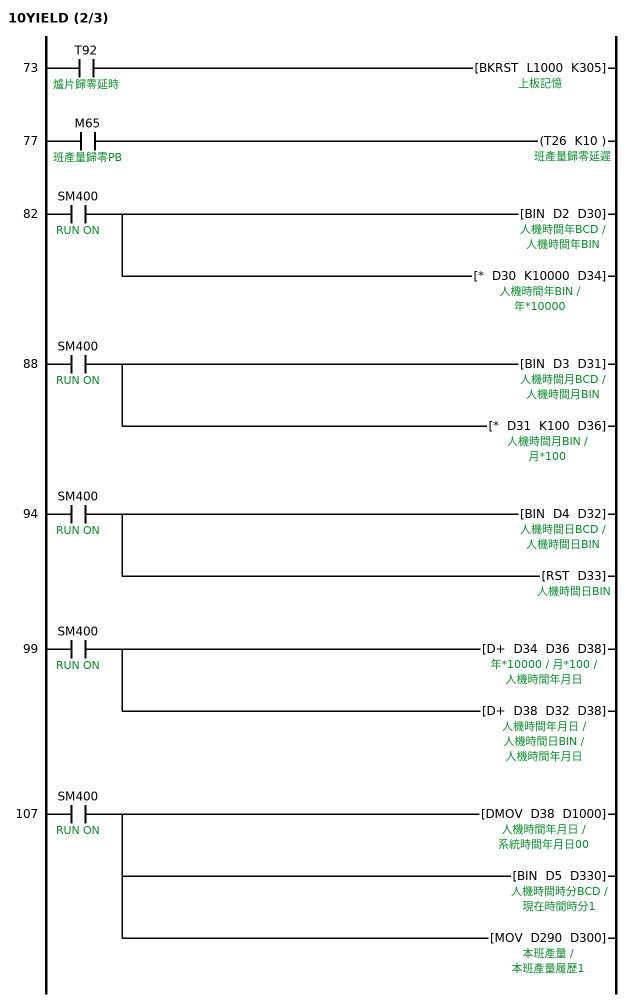
[picture p48: ladder of 10YIELD, rungs at steps 73 to 107]
73    LD      T92  ; 爐片歸零延時
      BKRST   L1000 K305
77    LD      M65  ; 班產量歸零PB
      OUT     T26 K10  ; 班產量歸零延遲
82    LD      SM400  ; RUN ON
      BIN     D2 D30  ; 人機時間年BCD / 人機時間年BIN
      *       D30 K10000 D34  ; 年*10000
88    LD      SM400  ; RUN ON
      BIN     D3 D31  ; 人機時間月BCD / 人機時間月BIN
      *       D31 K100 D36  ; 月*100
94    LD      SM400  ; RUN ON
      BIN     D4 D32  ; 人機時間日BCD / 人機時間日BIN
      RST     D33  ; 人機時間日BIN
99    LD      SM400  ; RUN ON
      D+      D34 D36 D38  ; 人機時間年月日
      D+      D38 D32 D38
107   LD      SM400  ; RUN ON
      DMOV    D38 D1000  ; 系統時間年月日00
      BIN     D5 D330  ; 人機時間時分BCD / 現在時間時分1
      MOV     D290 D300  ; 本班產量履歷1
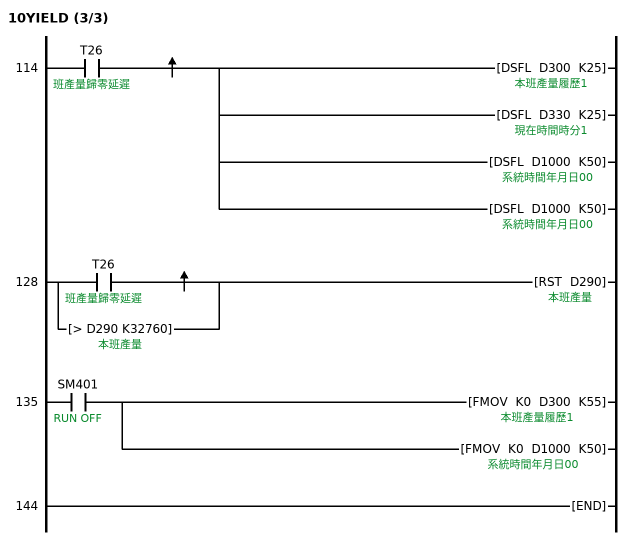
114   LD      T26  ; 班產量歸零延遲
      MEP
      DSFL    D300 K25
      DSFL    D330 K25
      DSFL    D1000 K50
      DSFL    D1000 K50
128   LD      T26  ; 班產量歸零延遲
      MEP
      OR>     D290 K32760  ; 本班產量
      RST     D290  ; 本班產量
135   LD      SM401  ; RUN OFF
      FMOV    K0 D300 K55
      FMOV    K0 D1000 K50
144   END
END_PROGRAM

PROGRAM 11MAINTE
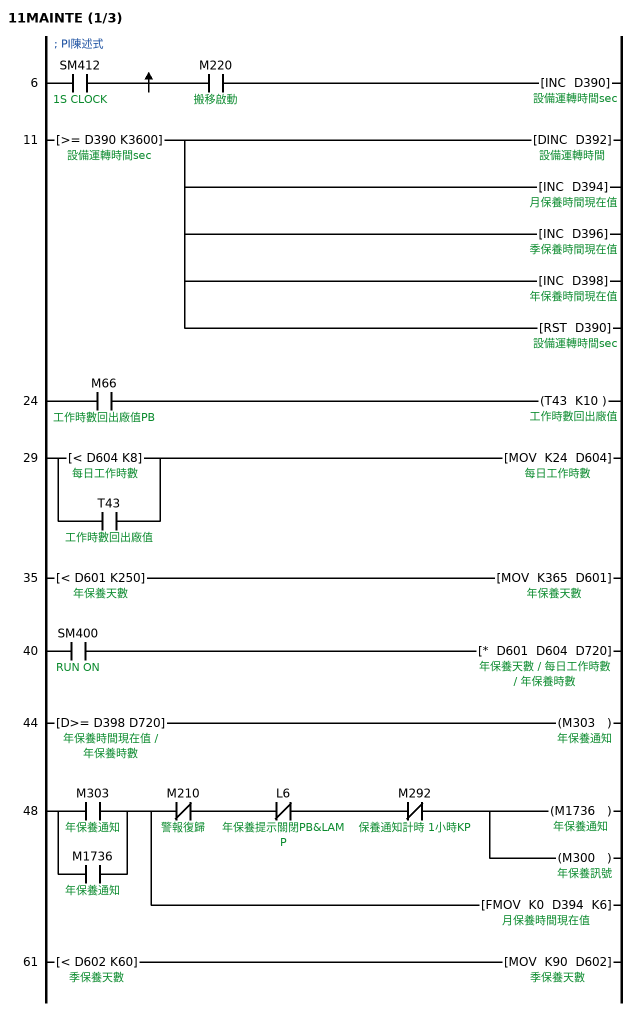
; PI陳述式
6     LD      SM412  ; 1S CLOCK
      MEP
      AND     M220  ; 搬移啟動
      INC     D390  ; 設備運轉時間sec
11    LD>=    D390 K3600  ; 設備運轉時間sec
      DINC    D392  ; 設備運轉時間
      INC     D394  ; 月保養時間現在值
      INC     D396  ; 季保養時間現在值
      INC     D398  ; 年保養時間現在值
      RST     D390  ; 設備運轉時間sec
24    LD      M66  ; 工作時數回出廠值PB
      OUT     T43 K10  ; 工作時數回出廠值
29    LD<     D604 K8  ; 每日工作時數
      OR      T43  ; 工作時數回出廠值
      MOV     K24 D604
35    LD<     D601 K250  ; 年保養天數
      MOV     K365 D601
40    LD      SM400  ; RUN ON
      *       D601 D604 D720  ; 年保養時數
44    LDD>=   D398 D720  ; 年保養時間現在值 / 年保養時數
      OUT     M303  ; 年保養通知
48    LD      M303  ; 年保養通知
      OR      M1736  ; 年保養通知
      MPS
      ANI     M210  ; 警報復歸
      ANI     L6  ; 年保養提示關閉PB&LAMP
      ANI     M292  ; 保養通知計時 1小時KP
      OUT     M1736  ; 年保養通知
      OUT     M300  ; 年保養訊號
      MPP
      FMOV    K0 D394 K6
61    LD<     D602 K60  ; 季保養天數
      MOV     K90 D602
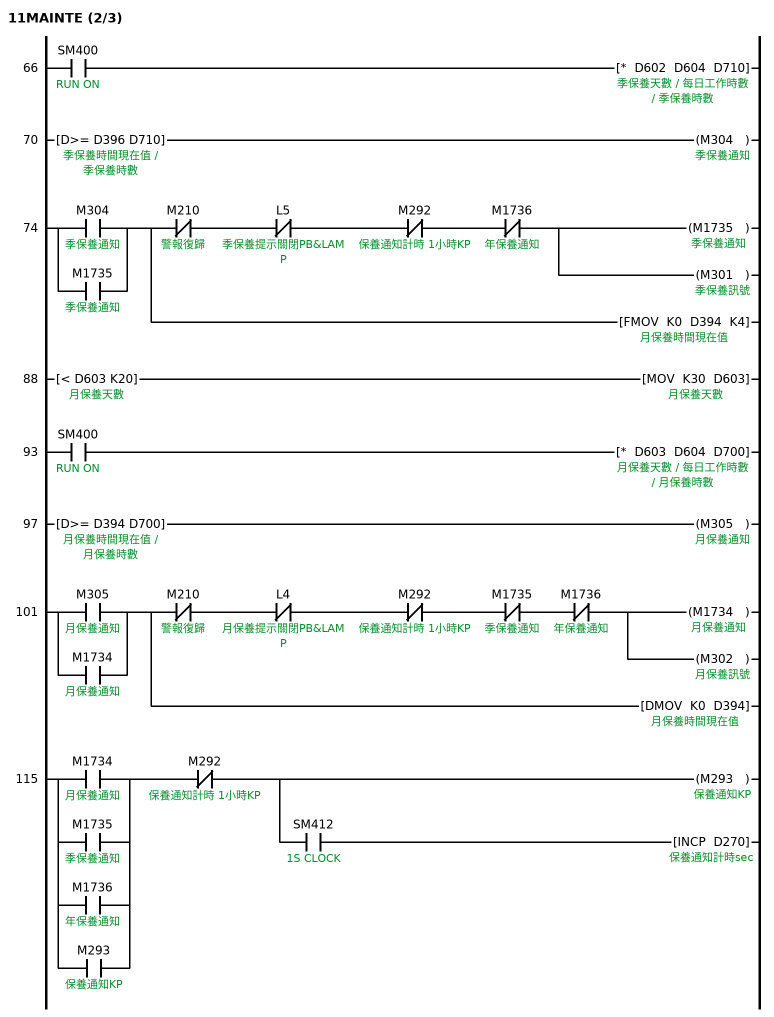
66    LD      SM400  ; RUN ON
      *       D602 D604 D710  ; 季保養時數
70    LDD>=   D396 D710  ; 季保養時間現在值 / 季保養時數
      OUT     M304  ; 季保養通知
74    LD      M304  ; 季保養通知
      OR      M1735  ; 季保養通知
      MPS
      ANI     M210  ; 警報復歸
      ANI     L5  ; 季保養提示關閉PB&LAMP
      ANI     M292  ; 保養通知計時 1小時KP
      ANI     M1736  ; 年保養通知
      OUT     M1735  ; 季保養通知
      OUT     M301  ; 季保養訊號
      MPP
      FMOV    K0 D394 K4
88    LD<     D603 K20  ; 月保養天數
      MOV     K30 D603
93    LD      SM400  ; RUN ON
      *       D603 D604 D700  ; 月保養時數
97    LDD>=   D394 D700  ; 月保養時間現在值 / 月保養時數
      OUT     M305  ; 月保養通知
101   LD      M305  ; 月保養通知
      OR      M1734  ; 月保養通知
      MPS
      ANI     M210  ; 警報復歸
      ANI     L4  ; 月保養提示關閉PB&LAMP
      ANI     M292  ; 保養通知計時 1小時KP
      ANI     M1735  ; 季保養通知
      ANI     M1736  ; 年保養通知
      OUT     M1734  ; 月保養通知
      OUT     M302  ; 月保養訊號
      MPP
      DMOV    K0 D394
115   LD      M1734  ; 月保養通知
      OR      M1735  ; 季保養通知
      OR      M1736  ; 年保養通知
      OR      M293  ; 保養通知KP
      ANI     M292  ; 保養通知計時 1小時KP
      OUT     M293  ; 保養通知KP
      AND     SM412  ; 1S CLOCK
      INCP    D270  ; 保養通知計時sec
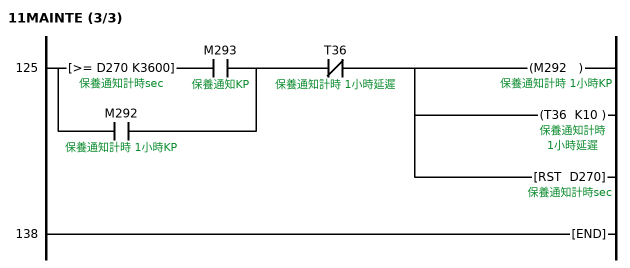
125   LD>=    D270 K3600  ; 保養通知計時sec
      AND     M293  ; 保養通知KP
      OR      M292  ; 保養通知計時 1小時KP
      ANI     T36  ; 保養通知計時 1小時延遲
      OUT     M292  ; 保養通知計時 1小時KP
      OUT     T36 K10  ; 保養通知計時 1小時延遲
      RST     D270  ; 保養通知計時sec
138   END
END_PROGRAM

PROGRAM 12ALARM1
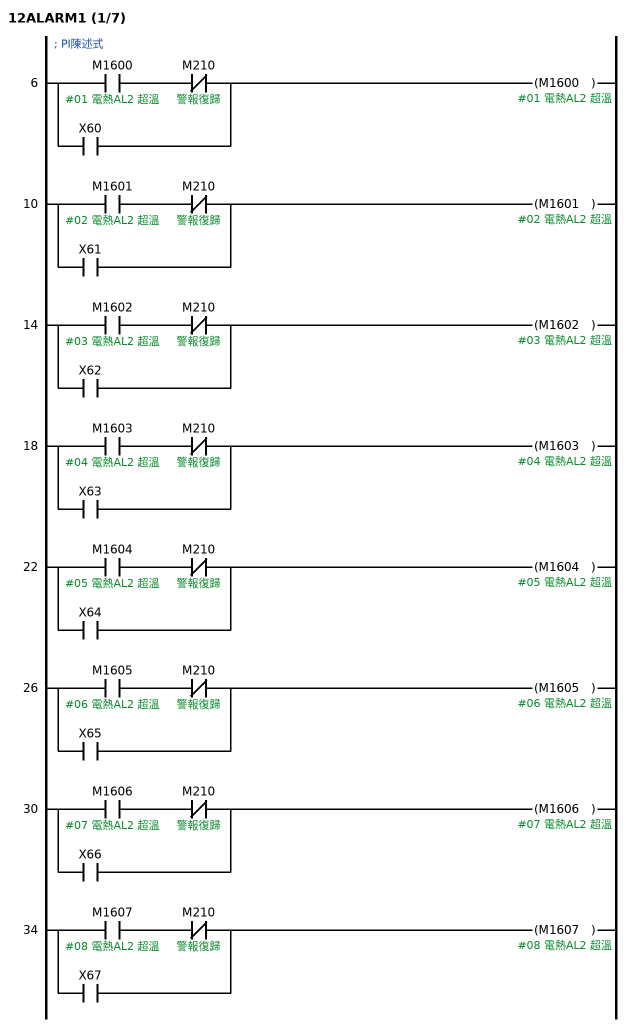
; PI陳述式
6     LD      M1600  ; #01 電熱AL2 超溫
      ANI     M210  ; 警報復歸
      OR      X60
      OUT     M1600  ; #01 電熱AL2 超溫
10    LD      M1601  ; #02 電熱AL2 超溫
      ANI     M210  ; 警報復歸
      OR      X61
      OUT     M1601  ; #02 電熱AL2 超溫
14    LD      M1602  ; #03 電熱AL2 超溫
      ANI     M210  ; 警報復歸
      OR      X62
      OUT     M1602  ; #03 電熱AL2 超溫
18    LD      M1603  ; #04 電熱AL2 超溫
      ANI     M210  ; 警報復歸
      OR      X63
      OUT     M1603  ; #04 電熱AL2 超溫
22    LD      M1604  ; #05 電熱AL2 超溫
      ANI     M210  ; 警報復歸
      OR      X64
      OUT     M1604  ; #05 電熱AL2 超溫
26    LD      M1605  ; #06 電熱AL2 超溫
      ANI     M210  ; 警報復歸
      OR      X65
      OUT     M1605  ; #06 電熱AL2 超溫
30    LD      M1606  ; #07 電熱AL2 超溫
      ANI     M210  ; 警報復歸
      OR      X66
      OUT     M1606  ; #07 電熱AL2 超溫
34    LD      M1607  ; #08 電熱AL2 超溫
      ANI     M210  ; 警報復歸
      OR      X67
      OUT     M1607  ; #08 電熱AL2 超溫
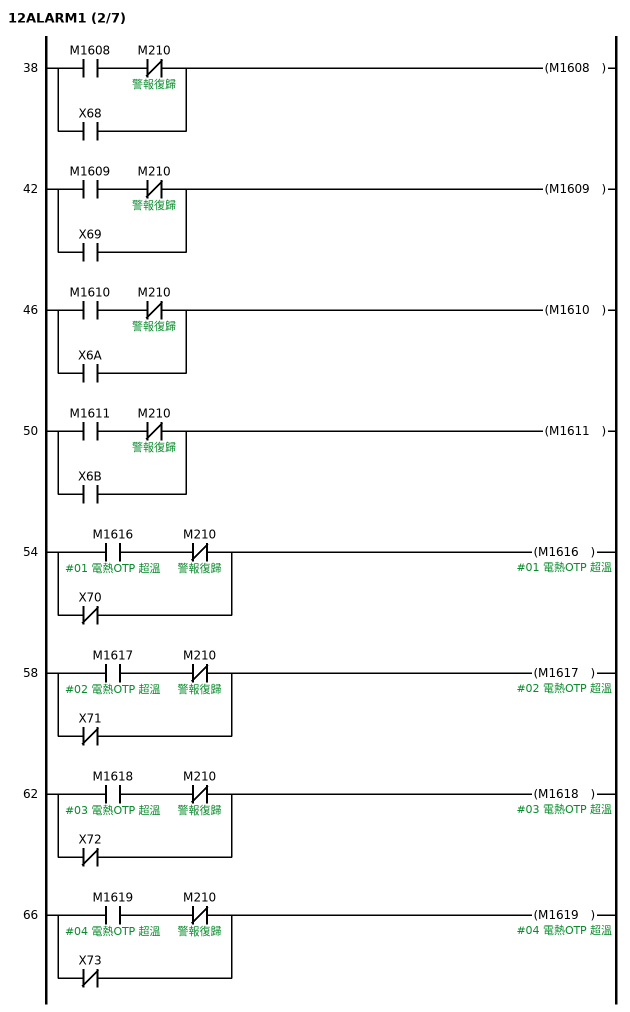
38    LD      M1608
      ANI     M210  ; 警報復歸
      OR      X68
      OUT     M1608
42    LD      M1609
      ANI     M210  ; 警報復歸
      OR      X69
      OUT     M1609
46    LD      M1610
      ANI     M210  ; 警報復歸
      OR      X6A
      OUT     M1610
50    LD      M1611
      ANI     M210  ; 警報復歸
      OR      X6B
      OUT     M1611
54    LD      M1616  ; #01 電熱OTP 超溫
      ANI     M210  ; 警報復歸
      ORI     X70
      OUT     M1616  ; #01 電熱OTP 超溫
58    LD      M1617  ; #02 電熱OTP 超溫
      ANI     M210  ; 警報復歸
      ORI     X71
      OUT     M1617  ; #02 電熱OTP 超溫
62    LD      M1618  ; #03 電熱OTP 超溫
      ANI     M210  ; 警報復歸
      ORI     X72
      OUT     M1618  ; #03 電熱OTP 超溫
66    LD      M1619  ; #04 電熱OTP 超溫
      ANI     M210  ; 警報復歸
      ORI     X73
      OUT     M1619  ; #04 電熱OTP 超溫
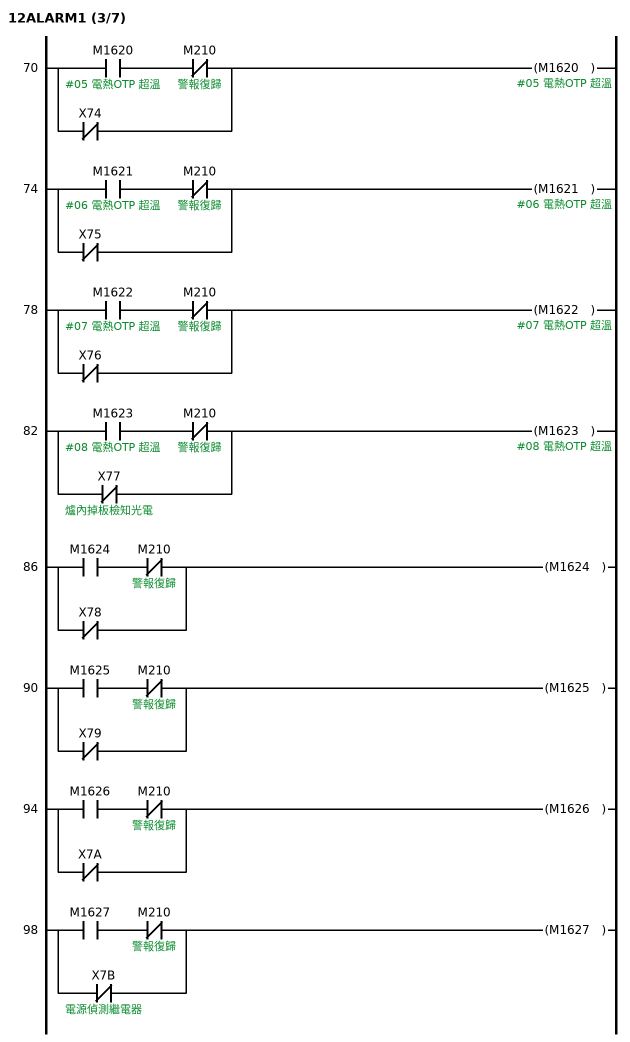
70    LD      M1620  ; #05 電熱OTP 超溫
      ANI     M210  ; 警報復歸
      ORI     X74
      OUT     M1620  ; #05 電熱OTP 超溫
74    LD      M1621  ; #06 電熱OTP 超溫
      ANI     M210  ; 警報復歸
      ORI     X75
      OUT     M1621  ; #06 電熱OTP 超溫
78    LD      M1622  ; #07 電熱OTP 超溫
      ANI     M210  ; 警報復歸
      ORI     X76
      OUT     M1622  ; #07 電熱OTP 超溫
82    LD      M1623  ; #08 電熱OTP 超溫
      ANI     M210  ; 警報復歸
      ORI     X77  ; 爐內掉板檢知光電
      OUT     M1623  ; #08 電熱OTP 超溫
86    LD      M1624
      ANI     M210  ; 警報復歸
      ORI     X78
      OUT     M1624
90    LD      M1625
      ANI     M210  ; 警報復歸
      ORI     X79
      OUT     M1625
94    LD      M1626
      ANI     M210  ; 警報復歸
      ORI     X7A
      OUT     M1626
98    LD      M1627
      ANI     M210  ; 警報復歸
      ORI     X7B  ; 電源偵測繼電器
      OUT     M1627
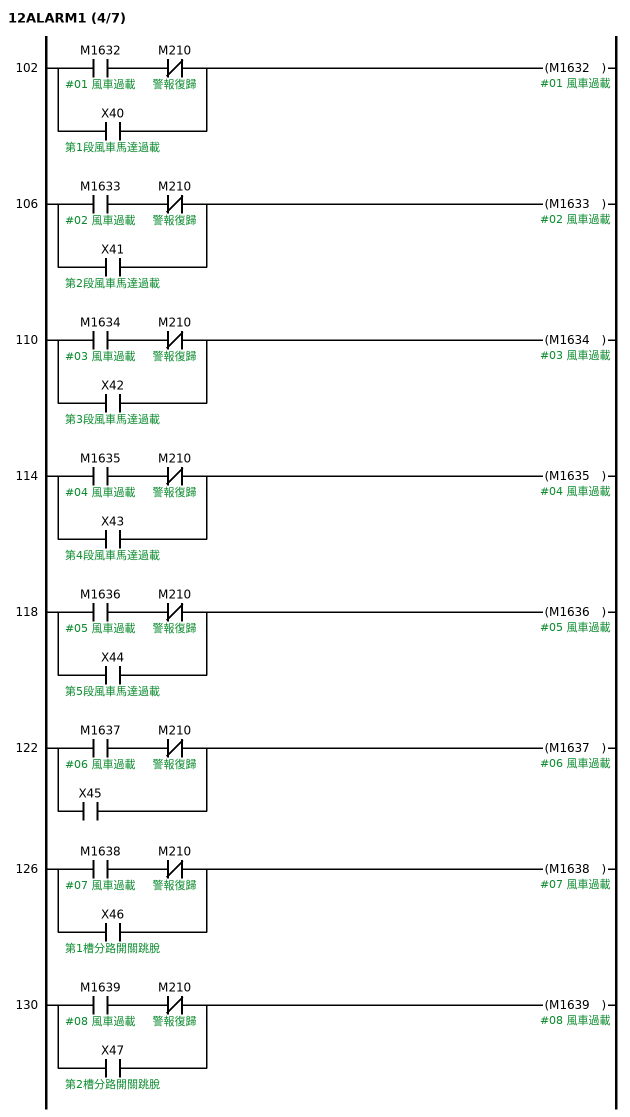
102   LD      M1632  ; #01 風車過載
      ANI     M210  ; 警報復歸
      OR      X40  ; 第1段風車馬達過載
      OUT     M1632  ; #01 風車過載
106   LD      M1633  ; #02 風車過載
      ANI     M210  ; 警報復歸
      OR      X41  ; 第2段風車馬達過載
      OUT     M1633  ; #02 風車過載
110   LD      M1634  ; #03 風車過載
      ANI     M210  ; 警報復歸
      OR      X42  ; 第3段風車馬達過載
      OUT     M1634  ; #03 風車過載
114   LD      M1635  ; #04 風車過載
      ANI     M210  ; 警報復歸
      OR      X43  ; 第4段風車馬達過載
      OUT     M1635  ; #04 風車過載
118   LD      M1636  ; #05 風車過載
      ANI     M210  ; 警報復歸
      OR      X44  ; 第5段風車馬達過載
      OUT     M1636  ; #05 風車過載
122   LD      M1637  ; #06 風車過載
      ANI     M210  ; 警報復歸
      OR      X45
      OUT     M1637  ; #06 風車過載
126   LD      M1638  ; #07 風車過載
      ANI     M210  ; 警報復歸
      OR      X46  ; 第1槽分路開關跳脫
      OUT     M1638  ; #07 風車過載
130   LD      M1639  ; #08 風車過載
      ANI     M210  ; 警報復歸
      OR      X47  ; 第2槽分路開關跳脫
      OUT     M1639  ; #08 風車過載
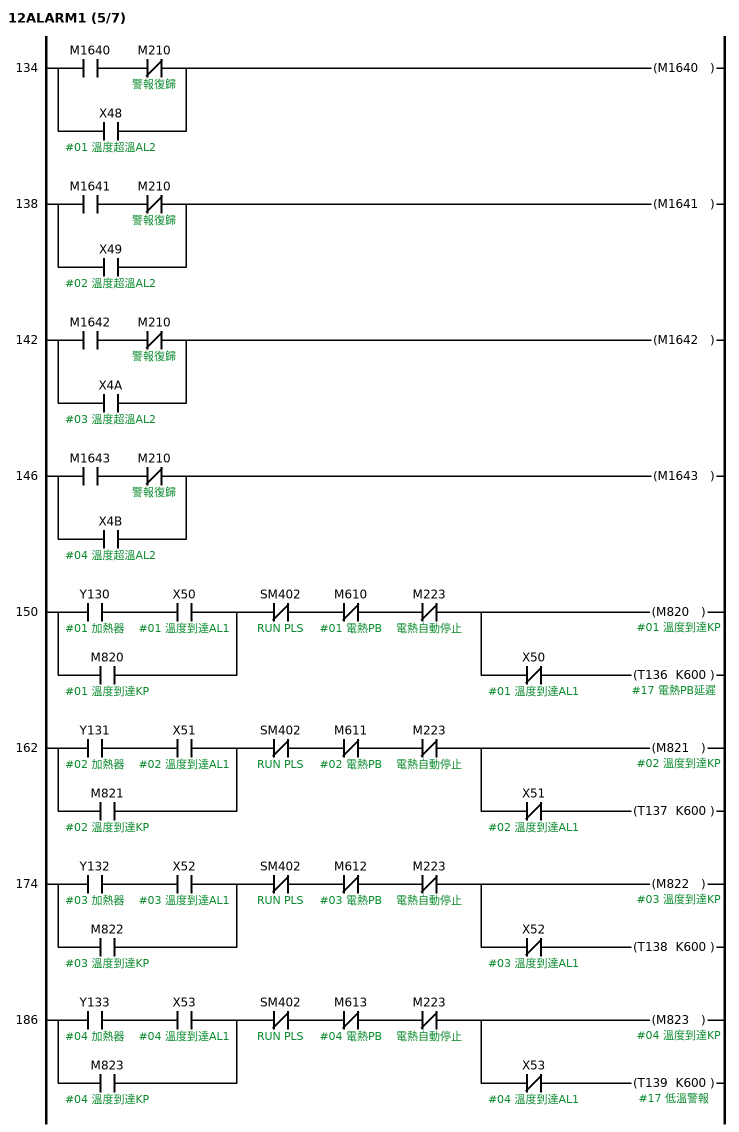
134   LD      M1640
      ANI     M210  ; 警報復歸
      OR      X48  ; #01 溫度超溫AL2
      OUT     M1640
138   LD      M1641
      ANI     M210  ; 警報復歸
      OR      X49  ; #02 溫度超溫AL2
      OUT     M1641
142   LD      M1642
      ANI     M210  ; 警報復歸
      OR      X4A  ; #03 溫度超溫AL2
      OUT     M1642
146   LD      M1643
      ANI     M210  ; 警報復歸
      OR      X4B  ; #04 溫度超溫AL2
      OUT     M1643
150   LD      Y130  ; #01 加熱器
      AND     X50  ; #01 溫度到達AL1
      OR      M820  ; #01 溫度到達KP
      ANI     SM402  ; RUN PLS
      ANI     M610  ; #01 電熱PB
      ANI     M223  ; 電熱自動停止
      OUT     M820  ; #01 溫度到達KP
      ANI     X50  ; #01 溫度到達AL1
      OUT     T136 K600  ; #17 電熱PB延遲
162   LD      Y131  ; #02 加熱器
      AND     X51  ; #02 溫度到達AL1
      OR      M821  ; #02 溫度到達KP
      ANI     SM402  ; RUN PLS
      ANI     M611  ; #02 電熱PB
      ANI     M223  ; 電熱自動停止
      OUT     M821  ; #02 溫度到達KP
      ANI     X51  ; #02 溫度到達AL1
      OUT     T137 K600
174   LD      Y132  ; #03 加熱器
      AND     X52  ; #03 溫度到達AL1
      OR      M822  ; #03 溫度到達KP
      ANI     SM402  ; RUN PLS
      ANI     M612  ; #03 電熱PB
      ANI     M223  ; 電熱自動停止
      OUT     M822  ; #03 溫度到達KP
      ANI     X52  ; #03 溫度到達AL1
      OUT     T138 K600
186   LD      Y133  ; #04 加熱器
      AND     X53  ; #04 溫度到達AL1
      OR      M823  ; #04 溫度到達KP
      ANI     SM402  ; RUN PLS
      ANI     M613  ; #04 電熱PB
      ANI     M223  ; 電熱自動停止
      OUT     M823  ; #04 溫度到達KP
      ANI     X53  ; #04 溫度到達AL1
      OUT     T139 K600  ; #17 低溫警報
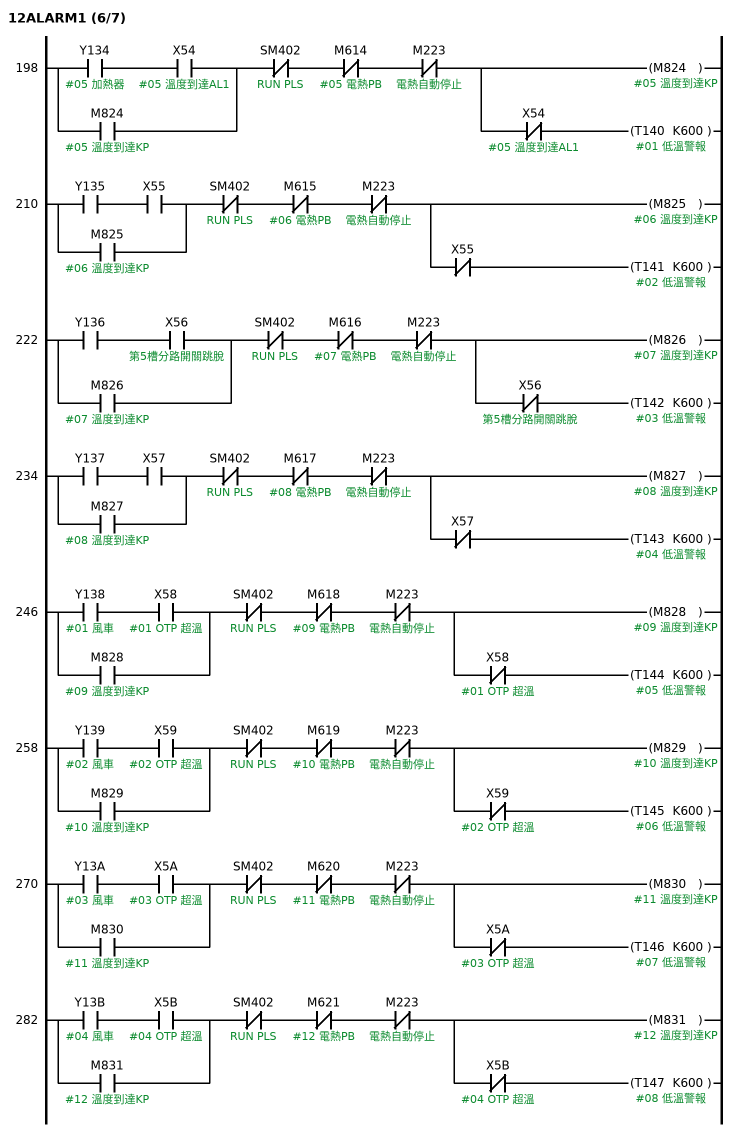
198   LD      Y134  ; #05 加熱器
      AND     X54  ; #05 溫度到達AL1
      OR      M824  ; #05 溫度到達KP
      ANI     SM402  ; RUN PLS
      ANI     M614  ; #05 電熱PB
      ANI     M223  ; 電熱自動停止
      OUT     M824  ; #05 溫度到達KP
      ANI     X54  ; #05 溫度到達AL1
      OUT     T140 K600  ; #01 低溫警報
210   LD      Y135
      AND     X55
      OR      M825  ; #06 溫度到達KP
      ANI     SM402  ; RUN PLS
      ANI     M615  ; #06 電熱PB
      ANI     M223  ; 電熱自動停止
      OUT     M825  ; #06 溫度到達KP
      ANI     X55
      OUT     T141 K600  ; #02 低溫警報
222   LD      Y136
      AND     X56  ; 第5槽分路開關跳脫
      OR      M826  ; #07 溫度到達KP
      ANI     SM402  ; RUN PLS
      ANI     M616  ; #07 電熱PB
      ANI     M223  ; 電熱自動停止
      OUT     M826  ; #07 溫度到達KP
      ANI     X56  ; 第5槽分路開關跳脫
      OUT     T142 K600  ; #03 低溫警報
234   LD      Y137
      AND     X57
      OR      M827  ; #08 溫度到達KP
      ANI     SM402  ; RUN PLS
      ANI     M617  ; #08 電熱PB
      ANI     M223  ; 電熱自動停止
      OUT     M827  ; #08 溫度到達KP
      ANI     X57
      OUT     T143 K600  ; #04 低溫警報
246   LD      Y138  ; #01 風車
      AND     X58  ; #01 OTP 超溫
      OR      M828  ; #09 溫度到達KP
      ANI     SM402  ; RUN PLS
      ANI     M618  ; #09 電熱PB
      ANI     M223  ; 電熱自動停止
      OUT     M828  ; #09 溫度到達KP
      ANI     X58  ; #01 OTP 超溫
      OUT     T144 K600  ; #05 低溫警報
258   LD      Y139  ; #02 風車
      AND     X59  ; #02 OTP 超溫
      OR      M829  ; #10 溫度到達KP
      ANI     SM402  ; RUN PLS
      ANI     M619  ; #10 電熱PB
      ANI     M223  ; 電熱自動停止
      OUT     M829  ; #10 溫度到達KP
      ANI     X59  ; #02 OTP 超溫
      OUT     T145 K600  ; #06 低溫警報
270   LD      Y13A  ; #03 風車
      AND     X5A  ; #03 OTP 超溫
      OR      M830  ; #11 溫度到達KP
      ANI     SM402  ; RUN PLS
      ANI     M620  ; #11 電熱PB
      ANI     M223  ; 電熱自動停止
      OUT     M830  ; #11 溫度到達KP
      ANI     X5A  ; #03 OTP 超溫
      OUT     T146 K600  ; #07 低溫警報
282   LD      Y13B  ; #04 風車
      AND     X5B  ; #04 OTP 超溫
      OR      M831  ; #12 溫度到達KP
      ANI     SM402  ; RUN PLS
      ANI     M621  ; #12 電熱PB
      ANI     M223  ; 電熱自動停止
      OUT     M831  ; #12 溫度到達KP
      ANI     X5B  ; #04 OTP 超溫
      OUT     T147 K600  ; #08 低溫警報
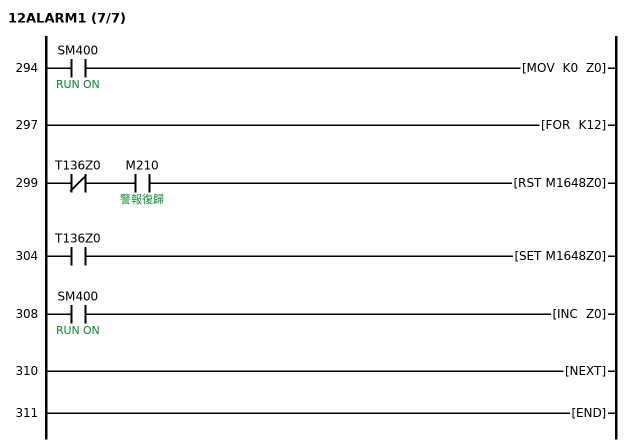
294   LD      SM400  ; RUN ON
      MOV     K0 Z0
297   FOR     K12
299   LDI     T136Z0
      AND     M210  ; 警報復歸
      RST     M1648Z0
304   LD      T136Z0
      SET     M1648Z0
308   LD      SM400  ; RUN ON
      INC     Z0
310   NEXT
311   END
END_PROGRAM

PROGRAM 13ALARM2
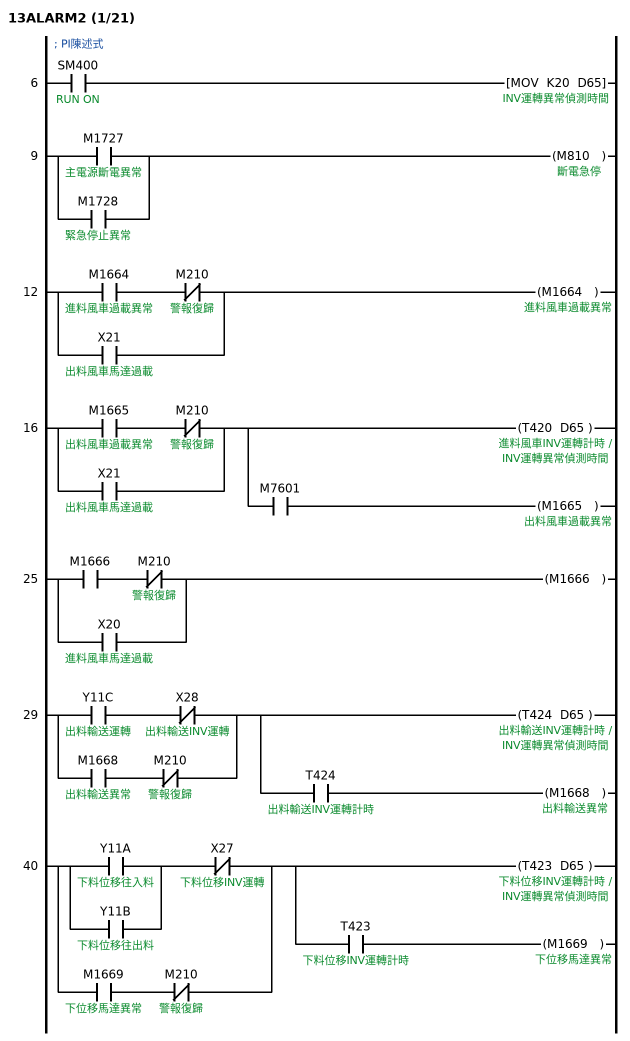
; PI陳述式
6     LD      SM400  ; RUN ON
      MOV     K20 D65  ; INV運轉異常偵測時間
9     LD      M1727  ; 主電源斷電異常
      OR      M1728  ; 緊急停止異常
      OUT     M810  ; 斷電急停
12    LD      M1664  ; 進料風車過載異常
      ANI     M210  ; 警報復歸
      OR      X21  ; 出料風車馬達過載
      OUT     M1664  ; 進料風車過載異常
16    LD      M1665  ; 出料風車過載異常
      ANI     M210  ; 警報復歸
      OR      X21  ; 出料風車馬達過載
      OUT     T420 D65  ; 進料風車INV運轉計時 / INV運轉異常偵測時間
      AND     M7601
      OUT     M1665  ; 出料風車過載異常
25    LD      M1666
      ANI     M210  ; 警報復歸
      OR      X20  ; 進料風車馬達過載
      OUT     M1666
29    LD      Y11C  ; 出料輸送運轉
      ANI     X28  ; 出料輸送INV運轉
      LD      M1668  ; 出料輸送異常
      ANI     M210  ; 警報復歸
      ORB
      OUT     T424 D65  ; 出料輸送INV運轉計時 / INV運轉異常偵測時間
      AND     T424  ; 出料輸送INV運轉計時
      OUT     M1668  ; 出料輸送異常
40    LD      Y11A  ; 下料位移往入料
      OR      Y11B  ; 下料位移往出料
      ANI     X27  ; 下料位移INV運轉
      LD      M1669  ; 下位移馬達異常
      ANI     M210  ; 警報復歸
      ORB
      OUT     T423 D65  ; 下料位移INV運轉計時 / INV運轉異常偵測時間
      AND     T423  ; 下料位移INV運轉計時
      OUT     M1669  ; 下位移馬達異常
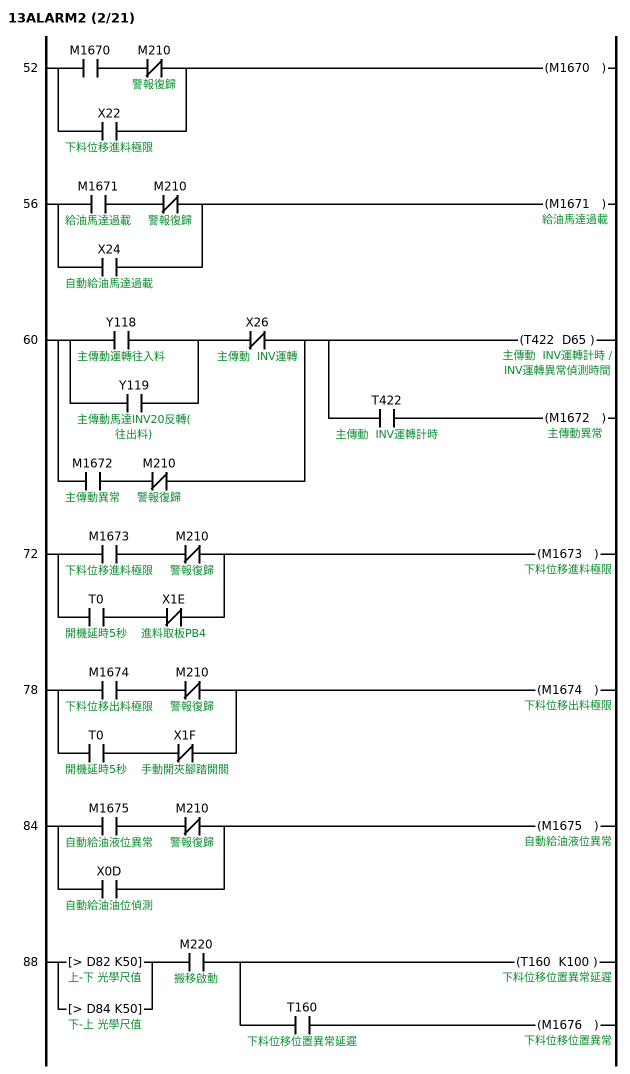
52    LD      M1670
      ANI     M210  ; 警報復歸
      OR      X22  ; 下料位移進料極限
      OUT     M1670
56    LD      M1671  ; 給油馬達過載
      ANI     M210  ; 警報復歸
      OR      X24  ; 自動給油馬達過載
      OUT     M1671  ; 給油馬達過載
60    LD      Y118  ; 主傳動運轉往入料
      OR      Y119  ; 主傳動馬達INV20反轉(往出料)
      ANI     X26  ; 主傳動  INV運轉
      LD      M1672  ; 主傳動異常
      ANI     M210  ; 警報復歸
      ORB
      OUT     T422 D65  ; 主傳動  INV運轉計時 / INV運轉異常偵測時間
      AND     T422  ; 主傳動  INV運轉計時
      OUT     M1672  ; 主傳動異常
72    LD      M1673  ; 下料位移進料極限
      ANI     M210  ; 警報復歸
      LD      T0  ; 開機延時5秒
      ANI     X1E  ; 進料取板PB4
      ORB
      OUT     M1673  ; 下料位移進料極限
78    LD      M1674  ; 下料位移出料極限
      ANI     M210  ; 警報復歸
      LD      T0  ; 開機延時5秒
      ANI     X1F  ; 手動開夾腳踏開關
      ORB
      OUT     M1674  ; 下料位移出料極限
84    LD      M1675  ; 自動給油液位異常
      ANI     M210  ; 警報復歸
      OR      X0D  ; 自動給油油位偵測
      OUT     M1675  ; 自動給油液位異常
88    LD>     D82 K50  ; 上-下 光學尺值
      OR>     D84 K50  ; 下-上 光學尺值
      AND     M220  ; 搬移啟動
      OUT     T160 K100  ; 下料位移位置異常延遲
      AND     T160  ; 下料位移位置異常延遲
      OUT     M1676  ; 下料位移位置異常
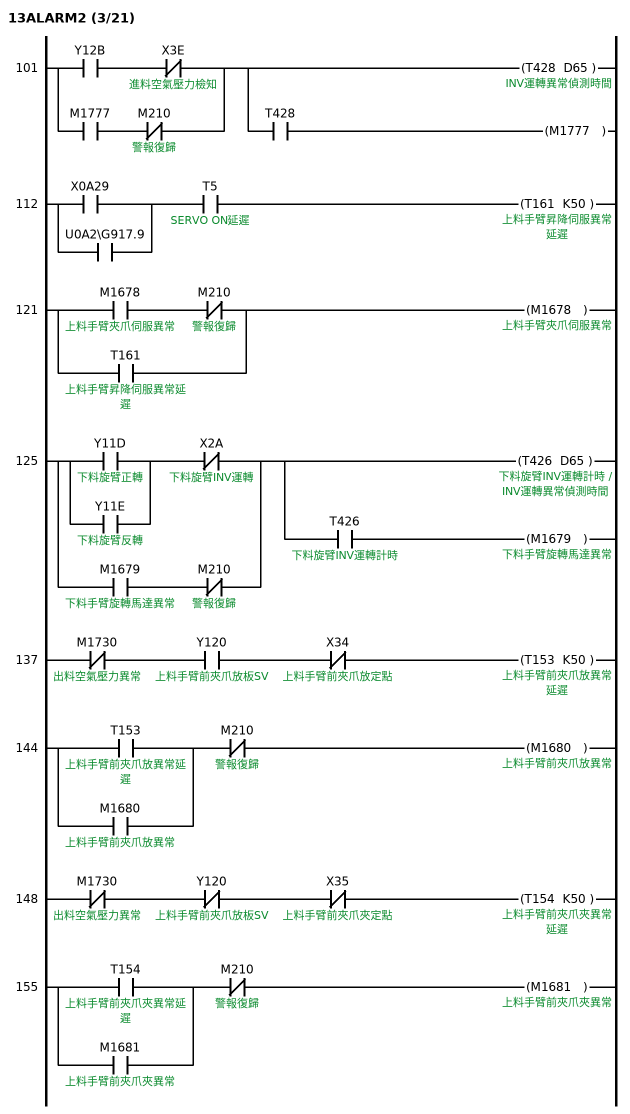
101   LD      Y12B
      ANI     X3E  ; 進料空氣壓力檢知
      LD      M1777
      ANI     M210  ; 警報復歸
      ORB
      OUT     T428 D65  ; INV運轉異常偵測時間
      AND     T428
      OUT     M1777
112   LD      X0A29
      OR      U0A2\G917.9
      AND     T5  ; SERVO ON延遲
      OUT     T161 K50  ; 上料手臂昇降伺服異常延遲
121   LD      M1678  ; 上料手臂夾爪伺服異常
      ANI     M210  ; 警報復歸
      OR      T161  ; 上料手臂昇降伺服異常延遲
      OUT     M1678  ; 上料手臂夾爪伺服異常
125   LD      Y11D  ; 下料旋臂正轉
      OR      Y11E  ; 下料旋臂反轉
      ANI     X2A  ; 下料旋臂INV運轉
      LD      M1679  ; 下料手臂旋轉馬達異常
      ANI     M210  ; 警報復歸
      ORB
      OUT     T426 D65  ; 下料旋臂INV運轉計時 / INV運轉異常偵測時間
      AND     T426  ; 下料旋臂INV運轉計時
      OUT     M1679  ; 下料手臂旋轉馬達異常
137   LDI     M1730  ; 出料空氣壓力異常
      AND     Y120  ; 上料手臂前夾爪放板SV
      ANI     X34  ; 上料手臂前夾爪放定點
      OUT     T153 K50  ; 上料手臂前夾爪放異常延遲
144   LD      T153  ; 上料手臂前夾爪放異常延遲
      OR      M1680  ; 上料手臂前夾爪放異常
      ANI     M210  ; 警報復歸
      OUT     M1680  ; 上料手臂前夾爪放異常
148   LDI     M1730  ; 出料空氣壓力異常
      ANI     Y120  ; 上料手臂前夾爪放板SV
      ANI     X35  ; 上料手臂前夾爪夾定點
      OUT     T154 K50  ; 上料手臂前夾爪夾異常延遲
155   LD      T154  ; 上料手臂前夾爪夾異常延遲
      OR      M1681  ; 上料手臂前夾爪夾異常
      ANI     M210  ; 警報復歸
      OUT     M1681  ; 上料手臂前夾爪夾異常
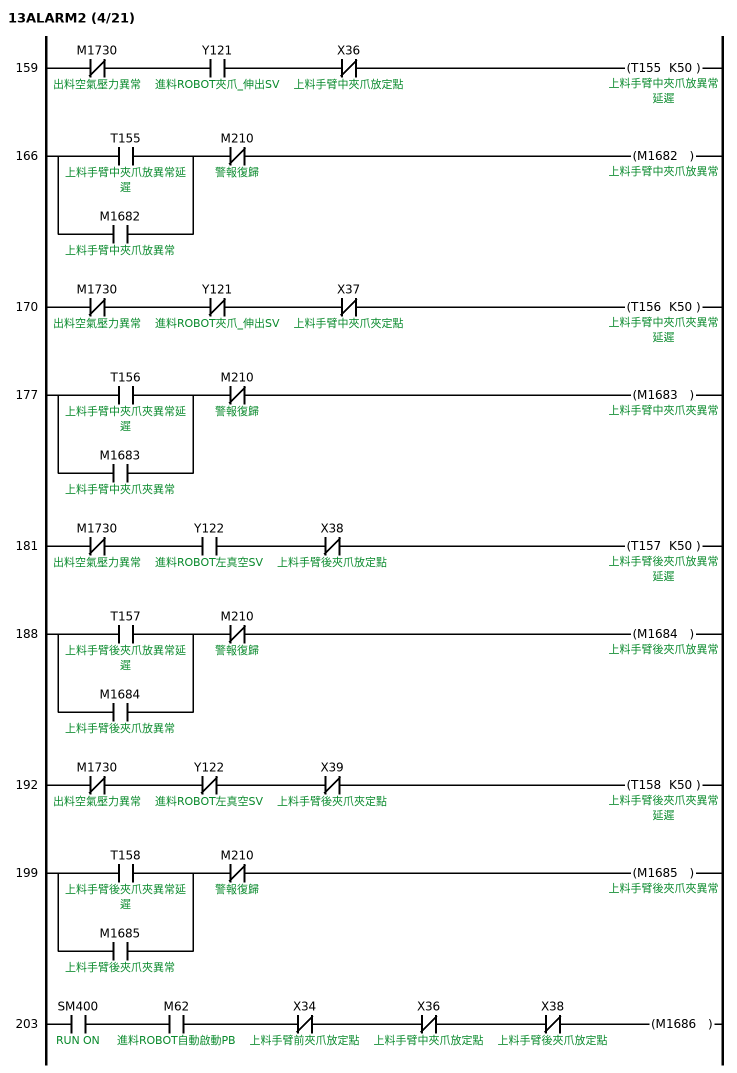
159   LDI     M1730  ; 出料空氣壓力異常
      AND     Y121  ; 進料ROBOT夾爪_伸出SV
      ANI     X36  ; 上料手臂中夾爪放定點
      OUT     T155 K50  ; 上料手臂中夾爪放異常延遲
166   LD      T155  ; 上料手臂中夾爪放異常延遲
      OR      M1682  ; 上料手臂中夾爪放異常
      ANI     M210  ; 警報復歸
      OUT     M1682  ; 上料手臂中夾爪放異常
170   LDI     M1730  ; 出料空氣壓力異常
      ANI     Y121  ; 進料ROBOT夾爪_伸出SV
      ANI     X37  ; 上料手臂中夾爪夾定點
      OUT     T156 K50  ; 上料手臂中夾爪夾異常延遲
177   LD      T156  ; 上料手臂中夾爪夾異常延遲
      OR      M1683  ; 上料手臂中夾爪夾異常
      ANI     M210  ; 警報復歸
      OUT     M1683  ; 上料手臂中夾爪夾異常
181   LDI     M1730  ; 出料空氣壓力異常
      AND     Y122  ; 進料ROBOT左真空SV
      ANI     X38  ; 上料手臂後夾爪放定點
      OUT     T157 K50  ; 上料手臂後夾爪放異常延遲
188   LD      T157  ; 上料手臂後夾爪放異常延遲
      OR      M1684  ; 上料手臂後夾爪放異常
      ANI     M210  ; 警報復歸
      OUT     M1684  ; 上料手臂後夾爪放異常
192   LDI     M1730  ; 出料空氣壓力異常
      ANI     Y122  ; 進料ROBOT左真空SV
      ANI     X39  ; 上料手臂後夾爪夾定點
      OUT     T158 K50  ; 上料手臂後夾爪夾異常延遲
199   LD      T158  ; 上料手臂後夾爪夾異常延遲
      OR      M1685  ; 上料手臂後夾爪夾異常
      ANI     M210  ; 警報復歸
      OUT     M1685  ; 上料手臂後夾爪夾異常
203   LD      SM400  ; RUN ON
      AND     M62  ; 進料ROBOT自動啟動PB
      ANI     X34  ; 上料手臂前夾爪放定點
      ANI     X36  ; 上料手臂中夾爪放定點
      ANI     X38  ; 上料手臂後夾爪放定點
      OUT     M1686
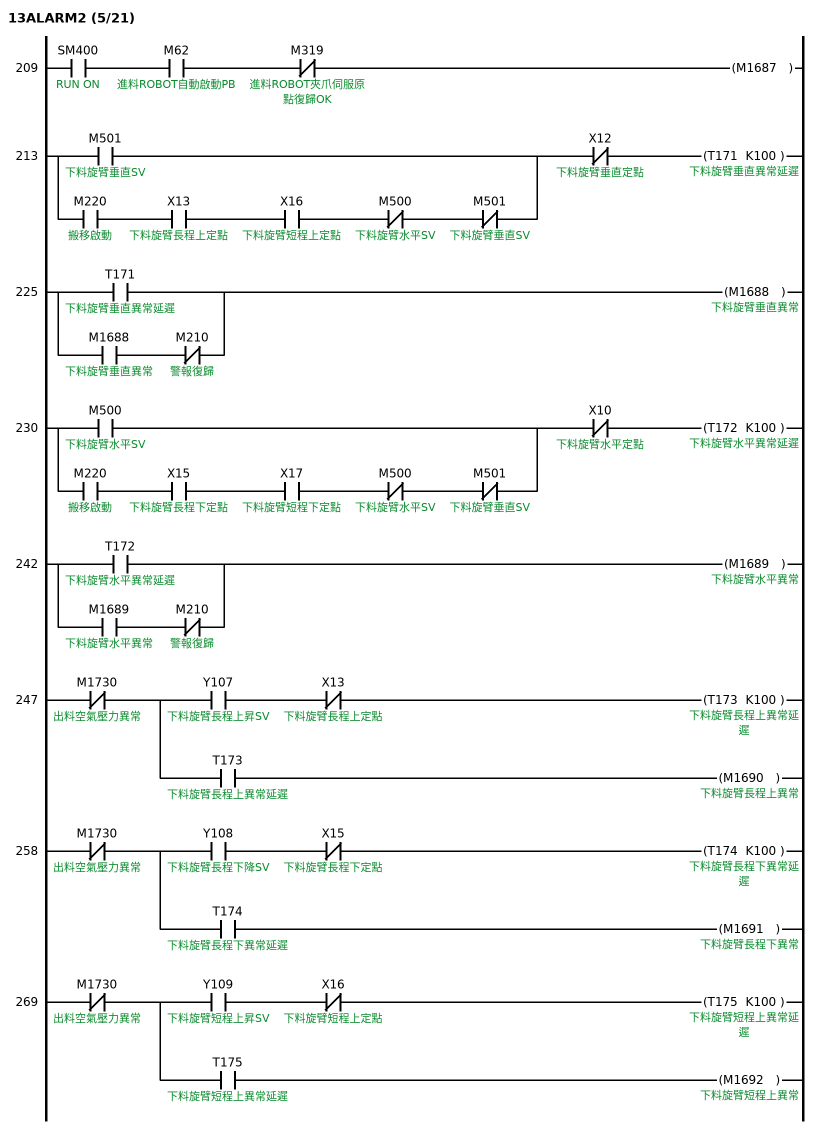
209   LD      SM400  ; RUN ON
      AND     M62  ; 進料ROBOT自動啟動PB
      ANI     M319  ; 進料ROBOT夾爪伺服原點復歸OK
      OUT     M1687
213   LD      M501  ; 下料旋臂垂直SV
      LD      M220  ; 搬移啟動
      AND     X13  ; 下料旋臂長程上定點
      AND     X16  ; 下料旋臂短程上定點
      ANI     M500  ; 下料旋臂水平SV
      ANI     M501  ; 下料旋臂垂直SV
      ORB
      ANI     X12  ; 下料旋臂垂直定點
      OUT     T171 K100  ; 下料旋臂垂直異常延遲
225   LD      T171  ; 下料旋臂垂直異常延遲
      LD      M1688  ; 下料旋臂垂直異常
      ANI     M210  ; 警報復歸
      ORB
      OUT     M1688  ; 下料旋臂垂直異常
230   LD      M500  ; 下料旋臂水平SV
      LD      M220  ; 搬移啟動
      AND     X15  ; 下料旋臂長程下定點
      AND     X17  ; 下料旋臂短程下定點
      ANI     M500  ; 下料旋臂水平SV
      ANI     M501  ; 下料旋臂垂直SV
      ORB
      ANI     X10  ; 下料旋臂水平定點
      OUT     T172 K100  ; 下料旋臂水平異常延遲
242   LD      T172  ; 下料旋臂水平異常延遲
      LD      M1689  ; 下料旋臂水平異常
      ANI     M210  ; 警報復歸
      ORB
      OUT     M1689  ; 下料旋臂水平異常
247   LDI     M1730  ; 出料空氣壓力異常
      MPS
      AND     Y107  ; 下料旋臂長程上昇SV
      ANI     X13  ; 下料旋臂長程上定點
      OUT     T173 K100  ; 下料旋臂長程上異常延遲
      MPP
      AND     T173  ; 下料旋臂長程上異常延遲
      OUT     M1690  ; 下料旋臂長程上異常
258   LDI     M1730  ; 出料空氣壓力異常
      MPS
      AND     Y108  ; 下料旋臂長程下降SV
      ANI     X15  ; 下料旋臂長程下定點
      OUT     T174 K100  ; 下料旋臂長程下異常延遲
      MPP
      AND     T174  ; 下料旋臂長程下異常延遲
      OUT     M1691  ; 下料旋臂長程下異常
269   LDI     M1730  ; 出料空氣壓力異常
      MPS
      AND     Y109  ; 下料旋臂短程上昇SV
      ANI     X16  ; 下料旋臂短程上定點
      OUT     T175 K100  ; 下料旋臂短程上異常延遲
      MPP
      AND     T175  ; 下料旋臂短程上異常延遲
      OUT     M1692  ; 下料旋臂短程上異常
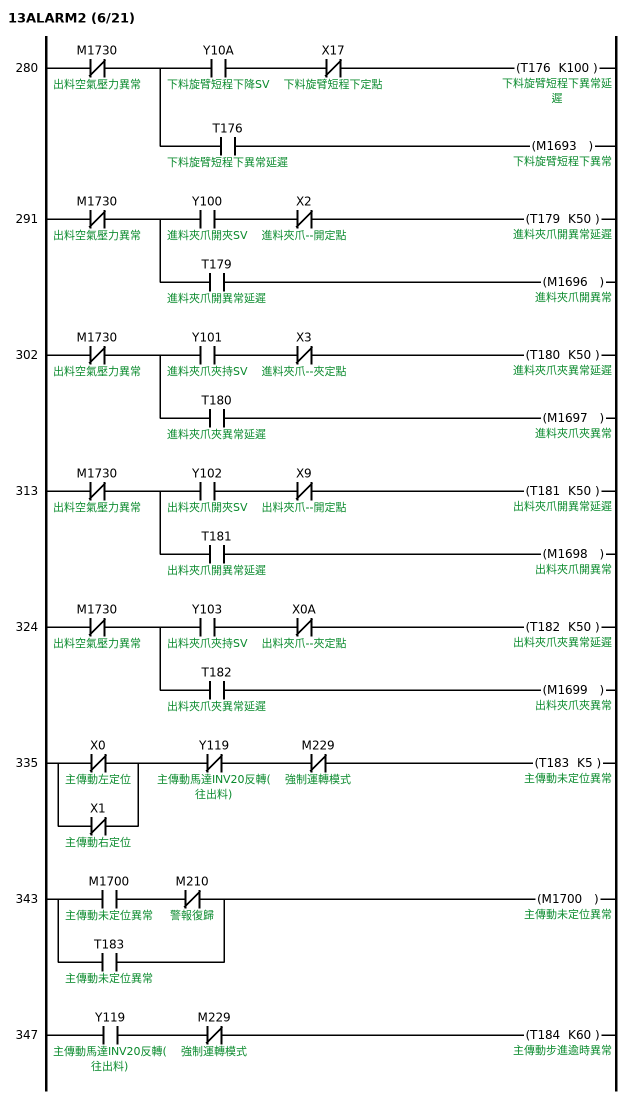
280   LDI     M1730  ; 出料空氣壓力異常
      MPS
      AND     Y10A  ; 下料旋臂短程下降SV
      ANI     X17  ; 下料旋臂短程下定點
      OUT     T176 K100  ; 下料旋臂短程下異常延遲
      MPP
      AND     T176  ; 下料旋臂短程下異常延遲
      OUT     M1693  ; 下料旋臂短程下異常
291   LDI     M1730  ; 出料空氣壓力異常
      MPS
      AND     Y100  ; 進料夾爪開夾SV
      ANI     X2  ; 進料夾爪--開定點
      OUT     T179 K50  ; 進料夾爪開異常延遲
      MPP
      AND     T179  ; 進料夾爪開異常延遲
      OUT     M1696  ; 進料夾爪開異常
302   LDI     M1730  ; 出料空氣壓力異常
      MPS
      AND     Y101  ; 進料夾爪夾持SV
      ANI     X3  ; 進料夾爪--夾定點
      OUT     T180 K50  ; 進料夾爪夾異常延遲
      MPP
      AND     T180  ; 進料夾爪夾異常延遲
      OUT     M1697  ; 進料夾爪夾異常
313   LDI     M1730  ; 出料空氣壓力異常
      MPS
      AND     Y102  ; 出料夾爪開夾SV
      ANI     X9  ; 出料夾爪--開定點
      OUT     T181 K50  ; 出料夾爪開異常延遲
      MPP
      AND     T181  ; 出料夾爪開異常延遲
      OUT     M1698  ; 出料夾爪開異常
324   LDI     M1730  ; 出料空氣壓力異常
      MPS
      AND     Y103  ; 出料夾爪夾持SV
      ANI     X0A  ; 出料夾爪--夾定點
      OUT     T182 K50  ; 出料夾爪夾異常延遲
      MPP
      AND     T182  ; 出料夾爪夾異常延遲
      OUT     M1699  ; 出料夾爪夾異常
335   LDI     X0  ; 主傳動左定位
      ORI     X1  ; 主傳動右定位
      ANI     Y119  ; 主傳動馬達INV20反轉(往出料)
      ANI     M229  ; 強制運轉模式
      OUT     T183 K5  ; 主傳動未定位異常
343   LD      M1700  ; 主傳動未定位異常
      ANI     M210  ; 警報復歸
      OR      T183  ; 主傳動未定位異常
      OUT     M1700  ; 主傳動未定位異常
347   LD      Y119  ; 主傳動馬達INV20反轉(往出料)
      ANI     M229  ; 強制運轉模式
      OUT     T184 K60  ; 主傳動步進逾時異常
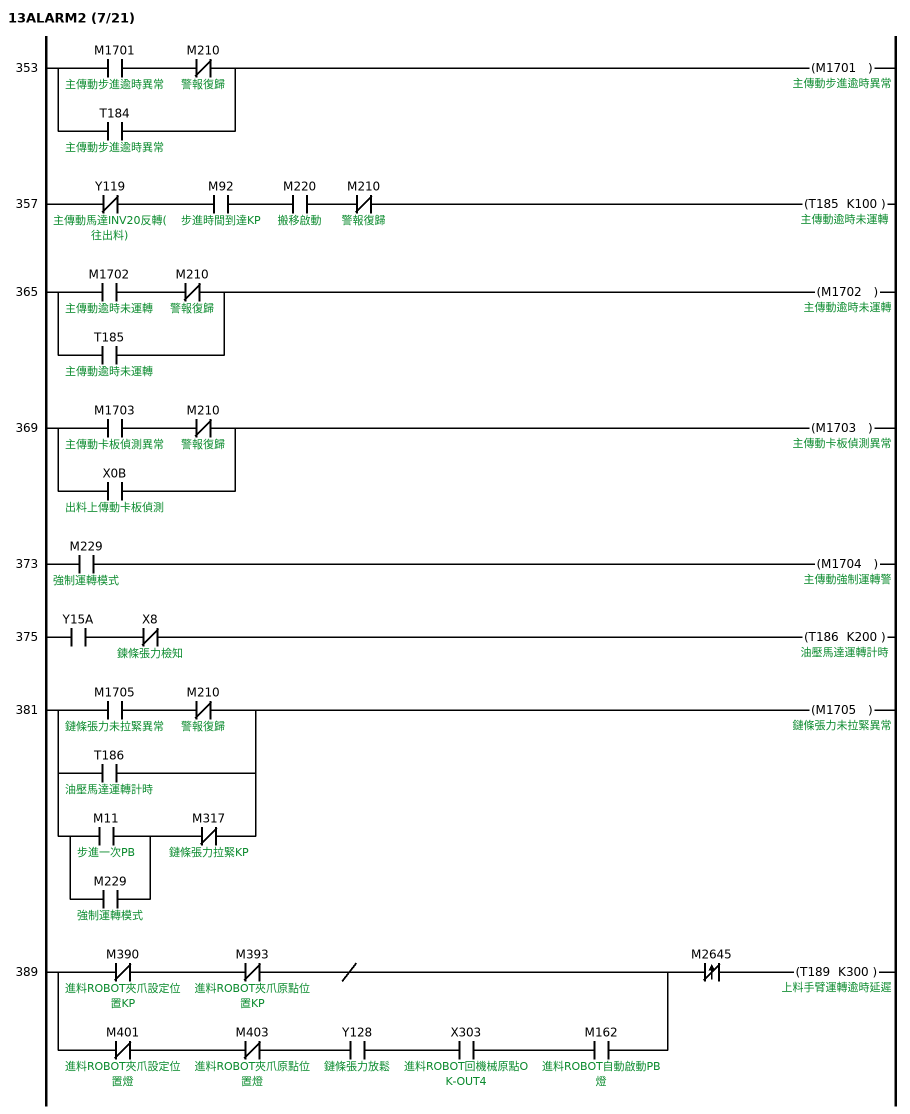
353   LD      M1701  ; 主傳動步進逾時異常
      ANI     M210  ; 警報復歸
      OR      T184  ; 主傳動步進逾時異常
      OUT     M1701  ; 主傳動步進逾時異常
357   LDI     Y119  ; 主傳動馬達INV20反轉(往出料)
      AND     M92  ; 步進時間到達KP
      AND     M220  ; 搬移啟動
      ANI     M210  ; 警報復歸
      OUT     T185 K100  ; 主傳動逾時未運轉
365   LD      M1702  ; 主傳動逾時未運轉
      ANI     M210  ; 警報復歸
      OR      T185  ; 主傳動逾時未運轉
      OUT     M1702  ; 主傳動逾時未運轉
369   LD      M1703  ; 主傳動卡板偵測異常
      ANI     M210  ; 警報復歸
      OR      X0B  ; 出料上傳動卡板偵測
      OUT     M1703  ; 主傳動卡板偵測異常
373   LD      M229  ; 強制運轉模式
      OUT     M1704  ; 主傳動強制運轉警
375   LD      Y15A
      ANI     X8  ; 鍊條張力檢知
      OUT     T186 K200  ; 油壓馬達運轉計時
381   LD      M1705  ; 鏈條張力未拉緊異常
      ANI     M210  ; 警報復歸
      OR      T186  ; 油壓馬達運轉計時
      LD      M11  ; 步進一次PB
      OR      M229  ; 強制運轉模式
      ANI     M317  ; 鏈條張力拉緊KP
      ORB
      OUT     M1705  ; 鏈條張力未拉緊異常
389   LDI     M390  ; 進料ROBOT夾爪設定位置KP
      ANI     M393  ; 進料ROBOT夾爪原點位置KP
      INV
      LDI     M401  ; 進料ROBOT夾爪設定位置燈
      ANI     M403  ; 進料ROBOT夾爪原點位置燈
      AND     Y128  ; 鏈條張力放鬆
      AND     X303  ; 進料ROBOT回機械原點OK-OUT4
      AND     M162  ; 進料ROBOT自動啟動PB燈
      ORB
      ANDPI   M2645
      OUT     T189 K300  ; 上料手臂運轉逾時延遲
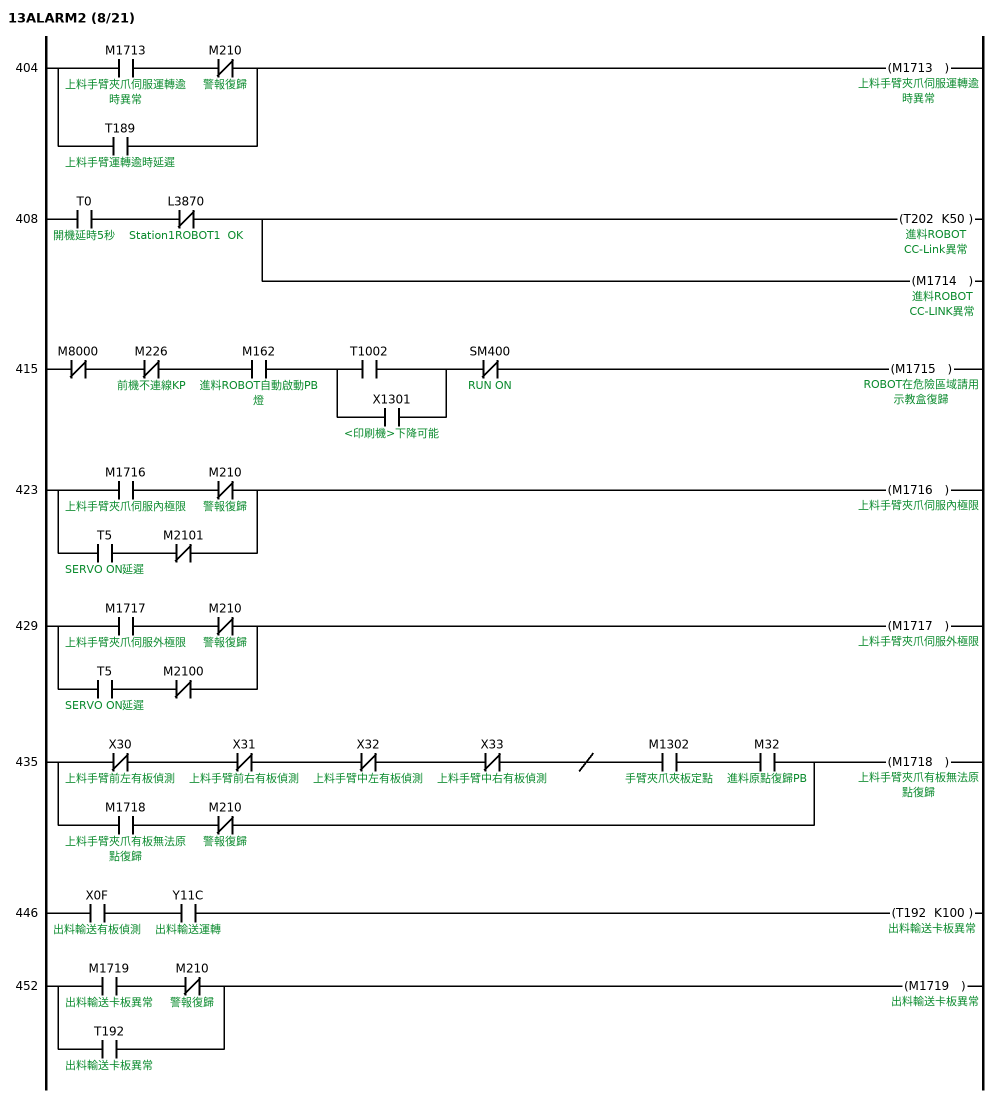
404   LD      M1713  ; 上料手臂夾爪伺服運轉逾時異常
      ANI     M210  ; 警報復歸
      OR      T189  ; 上料手臂運轉逾時延遲
      OUT     M1713  ; 上料手臂夾爪伺服運轉逾時異常
408   LD      T0  ; 開機延時5秒
      ANI     L3870  ; Station1ROBOT1  OK
      OUT     T202 K50  ; 進料ROBOT CC-Link異常
      OUT     M1714  ; 進料ROBOT CC-LINK異常
415   LDI     M8000
      ANI     M226  ; 前機不連線KP
      AND     M162  ; 進料ROBOT自動啟動PB燈
      LD      T1002
      OR      X1301  ; <印刷機>下降可能
      ANB
      ANI     SM400  ; RUN ON
      OUT     M1715  ; ROBOT在危險區域請用示教盒復歸
423   LD      M1716  ; 上料手臂夾爪伺服內極限
      ANI     M210  ; 警報復歸
      LD      T5  ; SERVO ON延遲
      ANI     M2101
      ORB
      OUT     M1716  ; 上料手臂夾爪伺服內極限
429   LD      M1717  ; 上料手臂夾爪伺服外極限
      ANI     M210  ; 警報復歸
      LD      T5  ; SERVO ON延遲
      ANI     M2100
      ORB
      OUT     M1717  ; 上料手臂夾爪伺服外極限
435   LDI     X30  ; 上料手臂前左有板偵測
      ANI     X31  ; 上料手臂前右有板偵測
      ANI     X32  ; 上料手臂中左有板偵測
      ANI     X33  ; 上料手臂中右有板偵測
      INV
      AND     M1302  ; 手臂夾爪夾板定點
      AND     M32  ; 進料原點復歸PB
      LD      M1718  ; 上料手臂夾爪有板無法原點復歸
      ANI     M210  ; 警報復歸
      ORB
      OUT     M1718  ; 上料手臂夾爪有板無法原點復歸
446   LD      X0F  ; 出料輸送有板偵測
      AND     Y11C  ; 出料輸送運轉
      OUT     T192 K100  ; 出料輸送卡板異常
452   LD      M1719  ; 出料輸送卡板異常
      ANI     M210  ; 警報復歸
      OR      T192  ; 出料輸送卡板異常
      OUT     M1719  ; 出料輸送卡板異常
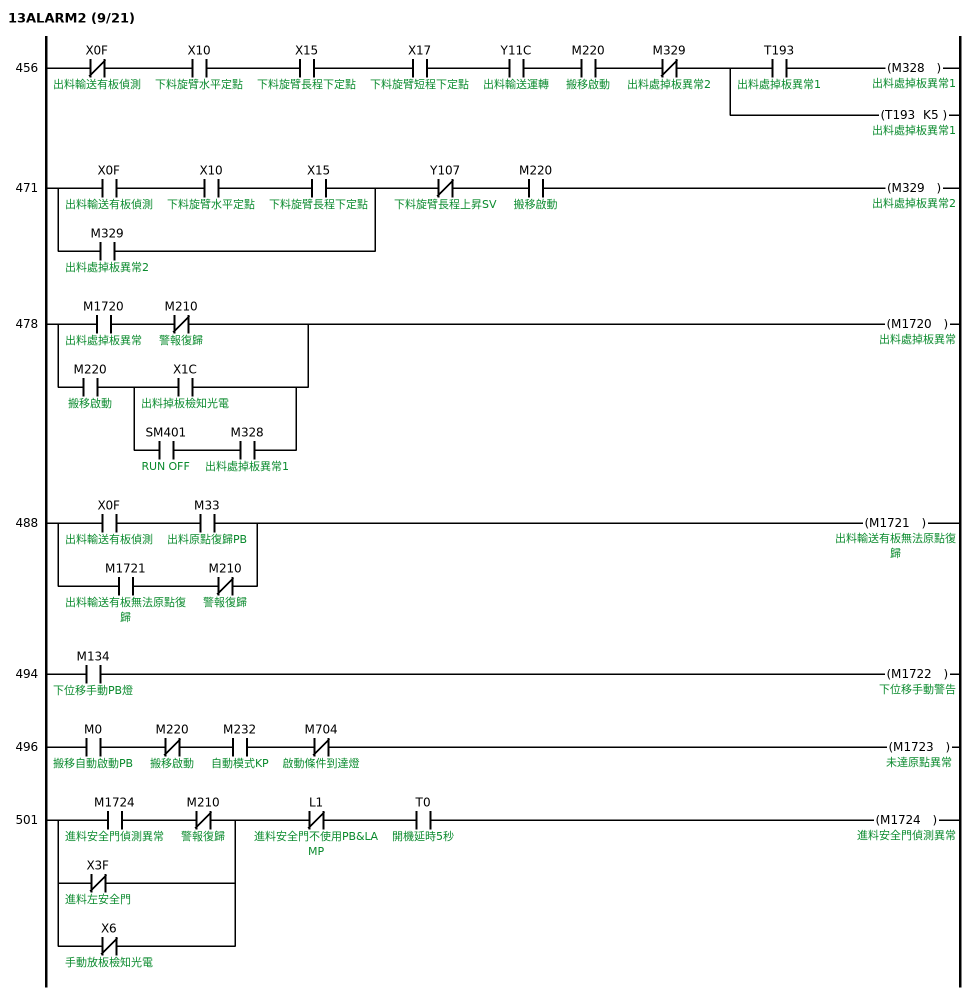
456   LDI     X0F  ; 出料輸送有板偵測
      AND     X10  ; 下料旋臂水平定點
      AND     X15  ; 下料旋臂長程下定點
      AND     X17  ; 下料旋臂短程下定點
      AND     Y11C  ; 出料輸送運轉
      AND     M220  ; 搬移啟動
      ANI     M329  ; 出料處掉板異常2
      MPS
      AND     T193  ; 出料處掉板異常1
      OUT     M328  ; 出料處掉板異常1
      MPP
      OUT     T193 K5  ; 出料處掉板異常1
471   LD      X0F  ; 出料輸送有板偵測
      AND     X10  ; 下料旋臂水平定點
      AND     X15  ; 下料旋臂長程下定點
      OR      M329  ; 出料處掉板異常2
      ANI     Y107  ; 下料旋臂長程上昇SV
      AND     M220  ; 搬移啟動
      OUT     M329  ; 出料處掉板異常2
478   LD      M1720  ; 出料處掉板異常
      ANI     M210  ; 警報復歸
      LD      M220  ; 搬移啟動
      LD      X1C  ; 出料掉板檢知光電
      LD      SM401  ; RUN OFF
      AND     M328  ; 出料處掉板異常1
      ORB
      ANB
      ORB
      OUT     M1720  ; 出料處掉板異常
488   LD      X0F  ; 出料輸送有板偵測
      AND     M33  ; 出料原點復歸PB
      LD      M1721  ; 出料輸送有板無法原點復歸
      ANI     M210  ; 警報復歸
      ORB
      OUT     M1721  ; 出料輸送有板無法原點復歸
494   LD      M134  ; 下位移手動PB燈
      OUT     M1722  ; 下位移手動警告
496   LD      M0  ; 搬移自動啟動PB
      ANI     M220  ; 搬移啟動
      AND     M232  ; 自動模式KP
      ANI     M704  ; 啟動條件到達燈
      OUT     M1723  ; 未達原點異常
501   LD      M1724  ; 進料安全門偵測異常
      ANI     M210  ; 警報復歸
      ORI     X3F  ; 進料左安全門
      ORI     X6  ; 手動放板檢知光電
      ANI     L1  ; 進料安全門不使用PB&LAMP
      AND     T0  ; 開機延時5秒
      OUT     M1724  ; 進料安全門偵測異常
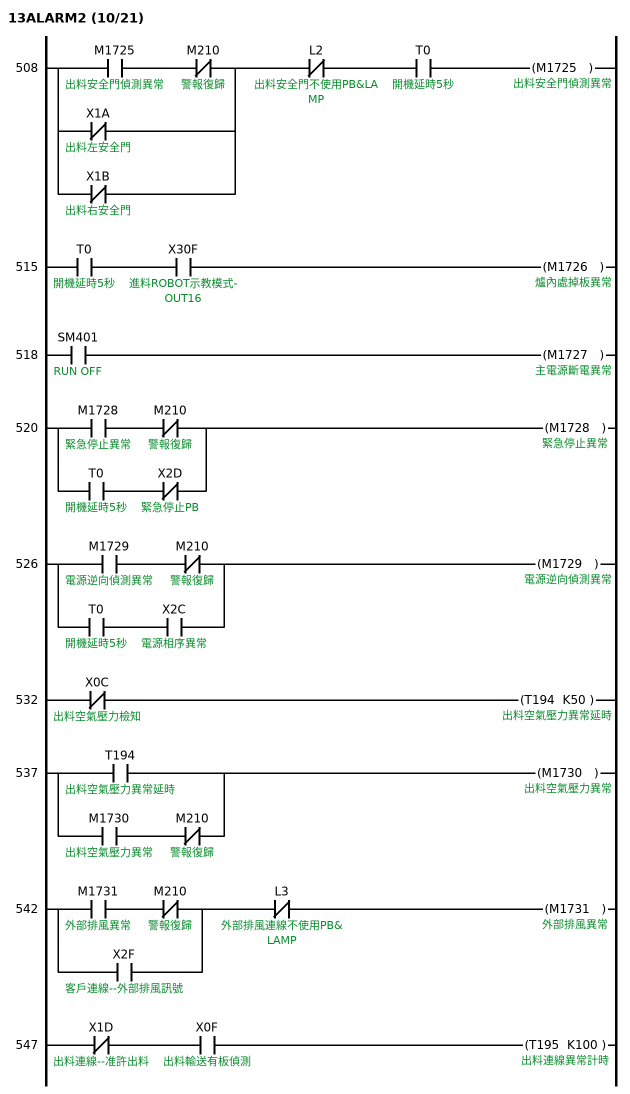
508   LD      M1725  ; 出料安全門偵測異常
      ANI     M210  ; 警報復歸
      ORI     X1A  ; 出料左安全門
      ORI     X1B  ; 出料右安全門
      ANI     L2  ; 出料安全門不使用PB&LAMP
      AND     T0  ; 開機延時5秒
      OUT     M1725  ; 出料安全門偵測異常
515   LD      T0  ; 開機延時5秒
      AND     X30F  ; 進料ROBOT示教模式-OUT16
      OUT     M1726  ; 爐內處掉板異常
518   LD      SM401  ; RUN OFF
      OUT     M1727  ; 主電源斷電異常
520   LD      M1728  ; 緊急停止異常
      ANI     M210  ; 警報復歸
      LD      T0  ; 開機延時5秒
      ANI     X2D  ; 緊急停止PB
      ORB
      OUT     M1728  ; 緊急停止異常
526   LD      M1729  ; 電源逆向偵測異常
      ANI     M210  ; 警報復歸
      LD      T0  ; 開機延時5秒
      AND     X2C  ; 電源相序異常
      ORB
      OUT     M1729  ; 電源逆向偵測異常
532   LDI     X0C  ; 出料空氣壓力檢知
      OUT     T194 K50  ; 出料空氣壓力異常延時
537   LD      T194  ; 出料空氣壓力異常延時
      LD      M1730  ; 出料空氣壓力異常
      ANI     M210  ; 警報復歸
      ORB
      OUT     M1730  ; 出料空氣壓力異常
542   LD      M1731  ; 外部排風異常
      ANI     M210  ; 警報復歸
      OR      X2F  ; 客戶連線--外部排風訊號
      ANI     L3  ; 外部排風連線不使用PB&LAMP
      OUT     M1731  ; 外部排風異常
547   LDI     X1D  ; 出料連線--准許出料
      AND     X0F  ; 出料輸送有板偵測
      OUT     T195 K100  ; 出料連線異常計時
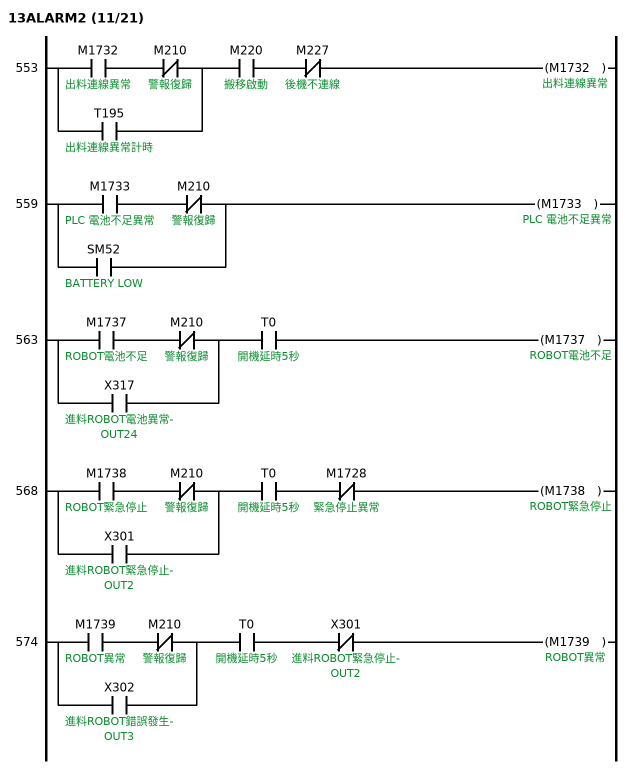
553   LD      M1732  ; 出料連線異常
      ANI     M210  ; 警報復歸
      OR      T195  ; 出料連線異常計時
      AND     M220  ; 搬移啟動
      ANI     M227  ; 後機不連線
      OUT     M1732  ; 出料連線異常
559   LD      M1733  ; PLC 電池不足異常
      ANI     M210  ; 警報復歸
      OR      SM52  ; BATTERY LOW
      OUT     M1733  ; PLC 電池不足異常
563   LD      M1737  ; ROBOT電池不足
      ANI     M210  ; 警報復歸
      OR      X317  ; 進料ROBOT電池異常-OUT24
      AND     T0  ; 開機延時5秒
      OUT     M1737  ; ROBOT電池不足
568   LD      M1738  ; ROBOT緊急停止
      ANI     M210  ; 警報復歸
      OR      X301  ; 進料ROBOT緊急停止-OUT2
      AND     T0  ; 開機延時5秒
      ANI     M1728  ; 緊急停止異常
      OUT     M1738  ; ROBOT緊急停止
574   LD      M1739  ; ROBOT異常
      ANI     M210  ; 警報復歸
      OR      X302  ; 進料ROBOT錯誤發生-OUT3
      AND     T0  ; 開機延時5秒
      ANI     X301  ; 進料ROBOT緊急停止-OUT2
      OUT     M1739  ; ROBOT異常
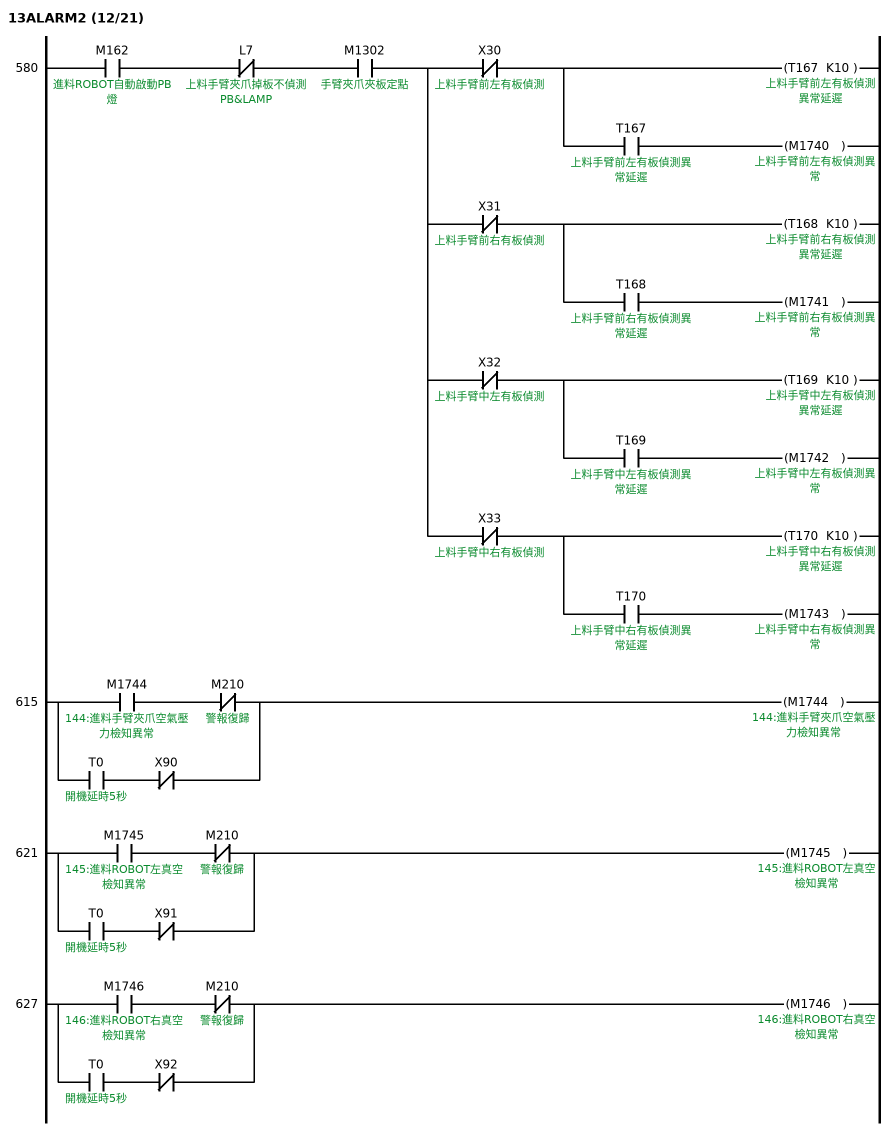
580   LD      M162  ; 進料ROBOT自動啟動PB燈
      ANI     L7  ; 上料手臂夾爪掉板不偵測PB&LAMP
      AND     M1302  ; 手臂夾爪夾板定點
      MPS
      ANI     X30  ; 上料手臂前左有板偵測
      OUT     T167 K10  ; 上料手臂前左有板偵測異常延遲
      AND     T167  ; 上料手臂前左有板偵測異常延遲
      OUT     M1740  ; 上料手臂前左有板偵測異常
      MRD
      ANI     X31  ; 上料手臂前右有板偵測
      OUT     T168 K10  ; 上料手臂前右有板偵測異常延遲
      AND     T168  ; 上料手臂前右有板偵測異常延遲
      OUT     M1741  ; 上料手臂前右有板偵測異常
      MRD
      ANI     X32  ; 上料手臂中左有板偵測
      OUT     T169 K10  ; 上料手臂中左有板偵測異常延遲
      AND     T169  ; 上料手臂中左有板偵測異常延遲
      OUT     M1742  ; 上料手臂中左有板偵測異常
      MPP
      ANI     X33  ; 上料手臂中右有板偵測
      OUT     T170 K10  ; 上料手臂中右有板偵測異常延遲
      AND     T170  ; 上料手臂中右有板偵測異常延遲
      OUT     M1743  ; 上料手臂中右有板偵測異常
615   LD      M1744  ; 144:進料手臂夾爪空氣壓力檢知異常
      ANI     M210  ; 警報復歸
      LD      T0  ; 開機延時5秒
      ANI     X90
      ORB
      OUT     M1744  ; 144:進料手臂夾爪空氣壓力檢知異常
621   LD      M1745  ; 145:進料ROBOT左真空檢知異常
      ANI     M210  ; 警報復歸
      LD      T0  ; 開機延時5秒
      ANI     X91
      ORB
      OUT     M1745  ; 145:進料ROBOT左真空檢知異常
627   LD      M1746  ; 146:進料ROBOT右真空檢知異常
      ANI     M210  ; 警報復歸
      LD      T0  ; 開機延時5秒
      ANI     X92
      ORB
      OUT     M1746  ; 146:進料ROBOT右真空檢知異常
